FUNCTION_BLOCK EL1018
VAR
	_io : EL1xx8_Data;
	{attribute addProperty Name "WcState"}
	_wcState : WcStateInputToggle;
	{attribute addProperty Name "Info data"}
	_infoData : InfoDataBase;
END_VAR

PROPERTY IO : REFERENCE TO EL1xx8_Data
GET
IO REF= _io;
END_GET
END_PROPERTY

PROPERTY WcState : REFERENCE TO WcStateInputToggle
GET
WcState REF= _wcState;
END_GET
END_PROPERTY

END_FUNCTION_BLOCK

(* stored: Version 1.1.0.1, ProductVersion 3.1.4024.9
   POU EL1018: Id {de4b66dc-047a-02af-2187-2d06206dc475}, SpecialFunc None
   Property IO: Id {fc6f60e0-fe67-06ef-36f1-c887e3dc4a86}
   Get Get: Id {9e319ab9-6fd0-0085-1b53-995273a171b5}
   Property WcState: Id {006e0ea8-d3e7-097f-2226-b6e7bf96472b}
   Get Get: Id {9dfec959-c246-06f2-2ef1-f0a3133e898f} *)
